FUNCTION_BLOCK FB4_Devices
VAR_INPUT
END_VAR
VAR_OUTPUT
END_VAR
VAR
END_VAR

//devices are not implemented for this project

END_FUNCTION_BLOCK

(* stored: Version 1.1.0.1, ProductVersion 3.1.4024.6
   POU FB4_Devices: Id {e2efe802-8b38-48d8-a591-337ee5822c42}, SpecialFunc None *)
